{attribute addProperty BoxType "EJ2521-0224-0016"}
{attribute addProperty Id "StatusAT %I*Status_F22324A31620Counter_valueAT %I*UINT16217Latch_valueAT %I*UINT16218"}
{attribute addProperty CRC "4194832074"}
{attribute addProperty SizeInBites "48"}
{attribute addProperty SizeInBytes "6"}
TYPE ENC_Status_compact_FA080ECA :
STRUCT
	{attribute addProperty Name "Status"}
	Status AT %I* : Status_F22324A3;
	{attribute addProperty Name "Counter_value"}
	Counter_value AT %I* : UINT;
	{attribute addProperty Name "Latch_value"}
	Latch_value AT %I* : UINT;
END_STRUCT
END_TYPE

(* stored: Version 1.2.0.0, ProductVersion 3.1.4024.9
   DUT ENC_Status_compact_FA080ECA: Id {91aeaac2-6b12-4435-90f5-460a34c10dd8} *)
